// TIA Portal project "Examen" (V16)

(* hardware
DEVICE "S71500/ET200MP station_1"  S7-1500 station
   slot 0: "Rail_0"  Rack  6ES7 590-1***0-0AA0
   slot 1: "PLC_1"  SIM-1500  6ES7 SIM-01500-APLC  V2.8
      slot 32768: "PROFINET interface_1"  X1
      slot 33024: "PROFINET interface_2"  X2
      slot 33280: "DP interface_1"  X4
   slot 2: "DI 32x24VDC HF_1"  DI 32x24VDC HF  6ES7 521-1BL00-0AB0  V2.2
   slot 3: "DQ 32x24VDC/0.5A HF_1"  DQ 32x24VDC/0.5A HF  6ES7 522-1BL01-0AB0  V1.1
   slot 4: "AI 8xU/I/RTD/TC ST_1"  AI 8xU/I/RTD/TC ST  6ES7 531-7KF00-0AB0  V2.2
   slot 5: "AQ 4xU/I ST_1"  AQ 4xU/I ST  6ES7 532-5HD00-0AB0  V2.2
DEVICE "HMI_1"  KTP700 Basic PN
   slot 0: "HMI_1"  KTP700 Basic PN  6AV2 123-2GB03-0AX0  16.0.0.0
   slot 1: "HMI_RT_1"  KTP700 Basic PN  6AV2 123-2GB03-0AX0  16.0.0.0
   slot 5: "HMI_1.IE_CP_1"  PROFINET Interface  16.0.0.0
      slot 1: "PROFINET Interface_1"  PROFINET Interface
         slot 1: "Port_1"  Port
*)

// ===== PLC "PLC_1"  SIM-1500 =====

VAR_GLOBAL   // PLC tag table "Default tag table"
   "LSH" AT %IW4 : Int;
   "Valor" AT %MD100 : Real;
   "Nivel_cm" AT %MW104 : Int;
   "Stop" AT %I0.0 : Bool;
   "Marcha" AT %I0.1 : Bool;
   "Lt-01" AT %I0.2 : Bool;
   "Nivel_op" AT %MW108 : Int;
   "Electrovalvula" AT %Q0.0 : Bool;
   "Bomba" AT %Q0.1 : Bool;
   "Limite_sup" AT %Q0.2 : Bool;
END_VAR

DATA_BLOCK "CONV_NIVEL_DB"   // DB1
{ S7_Optimized_Access := 'TRUE' }
VERSION : 0.1
// stored: InstanceOfName CONV_NIVEL
"CONV_NIVEL"
BEGIN
END_DATA_BLOCK

DATA_BLOCK "Programa_DB"   // DB2
{ S7_Optimized_Access := 'TRUE' }
VERSION : 0.1
// stored: InstanceOfName Programa
"Programa"
BEGIN
END_DATA_BLOCK

FUNCTION_BLOCK "CONV_NIVEL"   // FB1, LAD
{ S7_Optimized_Access := 'TRUE' }
VERSION : 0.1
   VAR_INPUT
      LSH : Int;
   END_VAR
   VAR_OUTPUT
      Nivel_cm : Int;
   END_VAR
   VAR
      LSH_NORM : Real;
   END_VAR
BEGIN

REGION Network 1
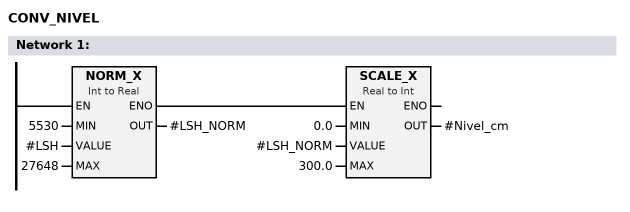
   RUNG wire#powerrail
      { S7_Templates := "[SrcType := Int, DestType := Real]" } Normalize(min := 5530, value := #LSH, max := 27648, out => #LSH_NORM)
      { S7_Templates := "[SrcType := Real, DestType := Int]" } Scale(min := 0.0, value := #LSH_NORM, max := 300.0, out => #Nivel_cm)
   END_RUNG
   // the same network as SCL:
   #LSH_NORM := NORM_X(MIN := 5530, VALUE := #LSH, MAX := 27648);
   #Nivel_cm := SCALE_X(MIN := 0.0, VALUE := #LSH_NORM, MAX := 300.0);
END_REGION
END_FUNCTION_BLOCK

FUNCTION_BLOCK "Programa"   // FB2, LAD
{ S7_Optimized_Access := 'TRUE' }
VERSION : 0.1
   VAR_INPUT
      STOP : Bool;
      MARCHA : Bool;
      "LT-01" : Bool;
      Nivel_sensado : Int;
      Nivel_operador : Int;
   END_VAR
   VAR_OUTPUT
      EV : Bool;
      "B-01" : Bool;
      Limit_Sup : Bool;
   END_VAR
   VAR
      M1 : Bool;
      M2 : Bool;
      M3 : Bool;
   END_VAR
BEGIN

REGION Network 1
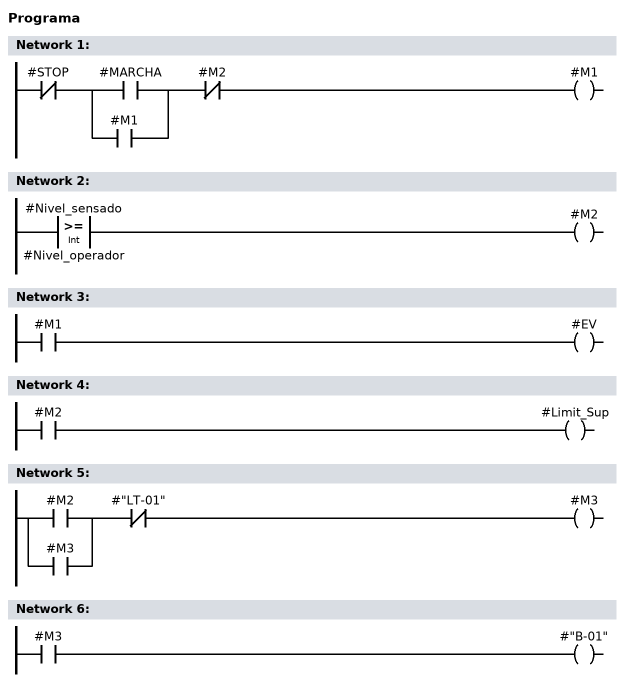
   RUNG wire#powerrail
      I_Contact( #STOP )
      wire#w1
      Contact( #MARCHA )
      wire#w2
      I_Contact( #M2 )
      Coil( #M1 )
   END_RUNG
   RUNG wire#w1
      Contact( #M1 )
   END_RUNG wire#w2
   // the same network as SCL:
   #M1 := NOT #STOP AND (#MARCHA OR #M1) AND NOT #M2;
END_REGION

REGION Network 2
   RUNG wire#powerrail
      { S7_Templates := "SrcType := Int" } GE_Contact(in1 := #Nivel_sensado, in2 := #Nivel_operador)
      Coil( #M2 )
   END_RUNG
   // the same network as SCL:
   #M2 := #Nivel_sensado >= #Nivel_operador;
END_REGION

REGION Network 3
   RUNG wire#powerrail
      Contact( #M1 )
      Coil( #EV )
   END_RUNG
   // the same network as SCL:
   #EV := #M1;
END_REGION

REGION Network 4
   RUNG wire#powerrail
      Contact( #M2 )
      Coil( #Limit_Sup )
   END_RUNG
   // the same network as SCL:
   #Limit_Sup := #M2;
END_REGION

REGION Network 5
   RUNG wire#powerrail
      Contact( #M2 )
      wire#w1
      I_Contact( #"LT-01" )
      Coil( #M3 )
   END_RUNG
   RUNG wire#powerrail
      Contact( #M3 )
   END_RUNG wire#w1
   // the same network as SCL:
   #M3 := (#M2 OR #M3) AND NOT #"LT-01";
END_REGION

REGION Network 6
   RUNG wire#powerrail
      Contact( #M3 )
      Coil( #"B-01" )
   END_RUNG
   // the same network as SCL:
   #"B-01" := #M3;
END_REGION
END_FUNCTION_BLOCK

ORGANIZATION_BLOCK "Main"   // OB1, LAD, ProgramCycle
TITLE = "Main Program Sweep (Cycle)"
{ S7_Optimized_Access := 'TRUE' }
VERSION : 0.1
   VAR_INPUT
      Initial_Call : Bool;   // Initial call of this OB
      Remanence : Bool;   // =True, if remanent data are available
   END_VAR
BEGIN

REGION Network 1
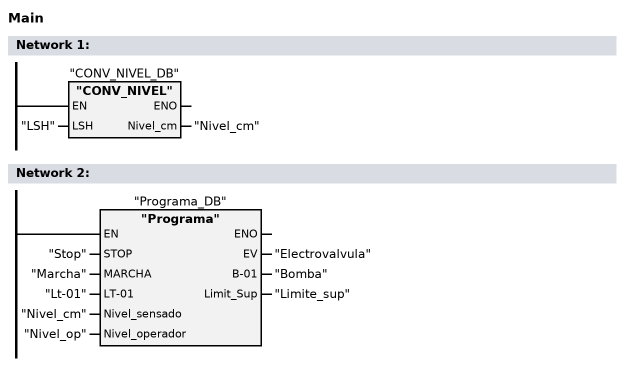
   RUNG wire#powerrail
      "CONV_NIVEL_DB"(LSH := "LSH", Nivel_cm => "Nivel_cm")
   END_RUNG
   // the same network as SCL:
   "CONV_NIVEL_DB"(LSH := "LSH", Nivel_cm => "Nivel_cm");   // "CONV_NIVEL"
END_REGION

REGION Network 2
   RUNG wire#powerrail
      "Programa_DB"(STOP := "Stop", MARCHA := "Marcha", "LT-01" := "Lt-01", Nivel_sensado := "Nivel_cm", Nivel_operador := "Nivel_op", EV => "Electrovalvula", "B-01" => "Bomba", Limit_Sup => "Limite_sup")
   END_RUNG
   // the same network as SCL:
   "Programa_DB"(STOP := "Stop",   // "Programa"
                 MARCHA := "Marcha",
                 "LT-01" := "Lt-01",
                 Nivel_sensado := "Nivel_cm",
                 Nivel_operador := "Nivel_op",
                 EV => "Electrovalvula",
                 "B-01" => "Bomba",
                 Limit_Sup => "Limite_sup");
END_REGION
END_ORGANIZATION_BLOCK

(* ===== HMI "HMI_RT_1" =====
system functions are stored by id; their names below are inferred from use
connection "HMI_Connection_1": ETHERNET, SMART_S7_1500_OMS

HMI tags "Default tag table"
   "Tag_ScreenNumber" : UInt, internal
   "Nivel_cm" : Int = PLC Nivel_cm AT %MW104, 1 s
   "Nivel_op" : Int = PLC Nivel_op AT %MW108, 1 s
   "Stop" : Bool = PLC Stop AT %I0.0, 1 s
   "Marcha" : Bool = PLC Marcha AT %I0.1, 1 s
   "Lt-01" : Bool = PLC "Lt-01" AT %I0.2, 1 s
   "Electrovalvula" : Bool = PLC Electrovalvula AT %Q0.0, 1 s
   "Bomba" : Bool = PLC Bomba AT %Q0.1, 1 s
   "Limite_sup" : Bool = PLC Limite_sup AT %Q0.2, 1 s

Template "Template_1" 800x480
   Button "Exit" at 714,429 size 71x50; TextOff 'Exit'; PictureOff "ExitRuntime_KTP700_Basic_PN_TR"; PictureOn "ExitRuntime_KTP700_Basic_PN_TR"
      on Release: StopRuntime(0)
   Button "Template_Button" at 614,429 size 71x50; TextOff 'Text'
   Button "Template_Button_1" at 514,429 size 71x50; TextOff 'Text'
   Button "Template_Button_2" at 414,429 size 71x50; TextOff 'Text'
   Button "Template_Button_3" at 314,429 size 71x50; TextOff 'Text'
   Button "Template_Button_4" at 214,429 size 71x50; TextOff 'Text'
   Button "Alarms" at 114,429 size 71x50; TextOff 'Alarms'; PictureOff "AlarmDisplay_KTP700_Basic_PN_TR"; PictureOn "AlarmDisplay_KTP700_Basic_PN_TR"
      on Release: function_ef3f5d25("Alarm window_Unacknowledged", -1)
   Button "Start screen" at 14,429 size 71x50; TextOff 'Start screen'; PictureOff "NavigateHome_KTP700_Basic_PN_TR"; PictureOn "NavigateHome_KTP700_Basic_PN_TR"
      on Release: ActivateScreen("Root screen", 0)
   SymbolicIOField "Symbolic_IO_Field_Screen" at 93,9 size 600x33; TextOff '0'; TextOn '1'; TextList "TextList_ScreenNames"
      ProcessValue <- "Tag_ScreenNumber"
      on Change: ActivateScreenByNumber("Tag_ScreenNumber", 0)
   DateTimeField "HmiScreenItemData" at 695,25 size 105x25
   DateTimeField "HmiScreenItemData_1" at 695,0 size 105x25
   GraphicView "Logo" at 0,0 size 91x51; Picture "Logo of HMI_1"

screen "Root screen" 800x480, template "Template_1"
   on GenerateScreen: SetTag("Tag_ScreenNumber", 1)
   TextField "HmiScreenItemData" at 80,225 size 640x25; Text 'Welcome to HMI_1 (KTP700 Basic+ PN)!'
   Button "HmiScreenItemData_1" at 36,87 size 159x47; TextOff 'System screens'; PictureOff "Navigates to System screens for KTP700 Basic+ PN 16.0.0.0"; PictureOn "Navigates to System screens for KTP700 Basic+ PN 16.0.0.0"
      on Release: ActivateScreen("System screens", 0)

screen "System screens" 800x480, template "Template_1"
   on GenerateScreen: SetTag("Tag_ScreenNumber", 2)
   Button "Back" at 1,52 size 159x47; TextOff 'Back'
      on Release: ActivateScreen("Root screen", 0)
   Button "HmiScreenItemData" at 36,146 size 159x47; TextOff 'Project information'; PictureOff "Navigates to Project information for KTP700 Basic+ PN 16.0.0.0"; PictureOn "Navigates to Project information for KTP700 Basic+ PN 16.0.0.0"
      on Release: ActivateScreen("Project information", 0)
   Button "HmiScreenItemData_1" at 36,205 size 159x47; TextOff 'User administration'; PictureOff "Navigates to User administration for KTP700 Basic+ PN 16.0.0.0"; PictureOn "Navigates to User administration for KTP700 Basic+ PN 16.0.0.0"
      on Release: ActivateScreen("User administration", 0)
   Button "HmiScreenItemData_2" at 36,264 size 159x47; TextOff 'System information'; PictureOff "Navigates to System information for KTP700 Basic+ PN 16.0.0.0"; PictureOn "Navigates to System information for KTP700 Basic+ PN 16.0.0.0"
      on Release: ActivateScreen("System information", 0)

screen "Project information" 800x480, template "Template_1"
   on GenerateScreen: SetTag("Tag_ScreenNumber", 3)
   TextField "HmiScreenItemData" at 35,102 size 171x28; Text 'Project name:'
   TextField "HmiScreenItemData_1" at 241,102 size 524x28; Text 'Examen'
   TextField "HmiScreenItemData_2" at 35,132 size 171x28; Text 'Created on:'
   TextField "HmiScreenItemData_3" at 241,132 size 524x28; Text '8/6/2023 9:55:00 PM'
   TextField "HmiScreenItemData_4" at 35,162 size 171x28; Text 'Author:'
   TextField "HmiScreenItemData_5" at 241,162 size 524x28; Text 'cepaq'
   TextField "HmiScreenItemData_6" at 35,192 size 171x28; Text 'Description:'
   TextField "HmiScreenItemData_7" at 241,192 size 524x28; Text '(not configured)'
   Button "Back" at 1,52 size 159x47; TextOff 'Back'
      on Release: ActivateScreen("System screens", 0)

screen "User administration" 800x480, template "Template_1"
   on GenerateScreen: SetTag("Tag_ScreenNumber", 4)
   UserView "HmiScreenItemData" at 1,100 size 796x321
   Button "Back" at 1,52 size 159x47; TextOff 'Back'
      on Release: ActivateScreen("System screens", 0)

screen "System information" 800x480, template "Template_1"
   on GenerateScreen: SetTag("Tag_ScreenNumber", 5)
   TextField "HmiScreenItemData" at 35,102 size 171x28; Text 'HMI device type:'
   TextField "HmiScreenItemData_1" at 241,102 size 524x28; Text 'KTP700 Basic+ PN 16.0.0.0'
   TextField "HmiScreenItemData_2" at 35,132 size 171x28; Text 'Connection:'
   TextField "HmiScreenItemData_3" at 241,132 size 524x28; Text 'PROFINET (X1)'
   TextField "HmiScreenItemData_4" at 35,162 size 171x28; Text 'PLC:'
   TextField "HmiScreenItemData_5" at 241,162 size 524x28; Text 'SIMATIC S7 1500'
   Button "Back" at 1,52 size 159x47; TextOff 'Back'
      on Release: ActivateScreen("System screens", 0)

screen "Proceso" 800x480
   TextField "Text field_1" at 280,36 size 240x23; Text 'Proceso de llenado y vaciado'
   Button "Button_1" at 70,106 size 96x32; TextOff 'Stop'
      Appearance <- "Stop"
   Button "Button_2" at 228,106 size 96x32; TextOff 'Start'
      Appearance <- "Marcha"
   IOField "I/O field_1" at 228,190 size 96x32; FormatPattern s999
      ProcessValue <- "Nivel_op"
   Bar "Bar_1" at 645,100 size 85x194; MinimumValue 0; MaximumValue 300
      ProcessValue <- "Nivel_cm"
   TextField "Text field_2" at 70,192 size 116x23; Text 'Setpoint (cm)'
   Circle "Circle_1" at 166,326 size 48x48
      Appearance <- "Electrovalvula"
   Circle "Circle_2" at 304,326 size 48x48
      Appearance <- "Bomba"
   Circle "Circle_3" at 453,326 size 48x48
      Appearance <- "Limite_sup"
   Circle "Circle_4" at 405,106 size 48x48
      Appearance <- "Lt-01"
   TextField "Text field_3" at 473,109 size 52x23; Text 'LT-01'
   TextField "Text field_4" at 419,386 size 128x23; Text 'Limite superior'
   TextField "Text field_5" at 635,71 size 108x23; Text 'Nivel tanque'
   TextField "Text field_6" at 175,386 size 26x23; Text 'EV'
   TextField "Text field_7" at 298,386 size 61x23; Text 'Bomba'
   GraphicView "Graphic view_1" at 280,254 size 116x65; Picture "Graphic_2"
*)